// TIA Portal V17 export
// export: Created 2023-02-25T16:31:53.0095529Z, ExportSetting WithDefaults, DisplayName Totally Integrated Automation Portal, DisplayVersion V17, DisplayName TIA Portal Openness, DisplayVersion V17, DisplayName TIA Portal Version Control Interface, DisplayVersion V17, DisplayName TIA Portal Test Suite Advanced, DisplayVersion V17, DisplayName STEP 7 Professional, DisplayVersion V17, DisplayName SIMATIC Energy Suite, DisplayVersion V17, DisplayName STEP 7 Safety, DisplayVersion V17, DisplayName WinCC Professional, DisplayVersion V17
FUNCTION "LOG_Light" : Void   // FC11, LAD
{ S7_Optimized_Access := 'TRUE' }
VERSION : 0.1
// stored: AutoNumber true, IsIECCheckEnabled false, SetENOAutomatically false, UDAEnableTagReadback false
BEGIN

REGION Network 1: Call: ButtonsLight
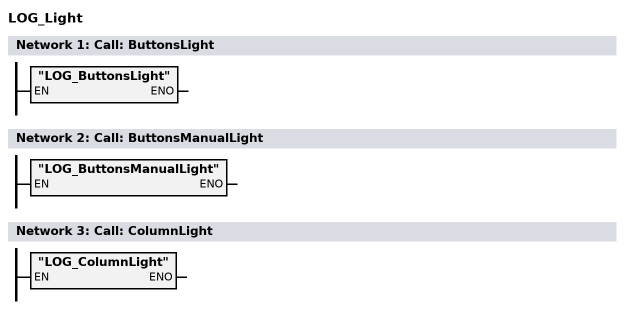
   RUNG wire#powerrail
      "LOG_ButtonsLight"()
   END_RUNG
   // the same network as SCL:
   "LOG_ButtonsLight"();
END_REGION

REGION Network 2: Call: ButtonsManualLight
   RUNG wire#powerrail
      "LOG_ButtonsManualLight"()
   END_RUNG
   // the same network as SCL:
   "LOG_ButtonsManualLight"();
END_REGION

REGION Network 3: Call: ColumnLight
   RUNG wire#powerrail
      "LOG_ColumnLight"()
   END_RUNG
   // the same network as SCL:
   "LOG_ColumnLight"();
END_REGION
END_FUNCTION
